Universal Robots PolyScope program: shot_03_120.urp

Program shot_03_120 (installation=default createdIn=5.11.11 lastSavedIn=5.11.11)
Robot Program (runOnlyOnce=true)
  Script file shot_03_120.script
    | def Program():
    |   CameraTcp = p[0.035, 0, 0.11, 1.2092, 1.2092, 1.2092]
    |   CameraWeight = 2
    |   CameraCog = [0.035, 0, 0.11]
    |   DefaultSpeed = 0.1
    |   DefaultZone = 0
    |   popup("Press 'Continue' to reset to Pose 0.", title="Ready?", blocking=True)
    |   set_tcp(CameraTcp)
    |   set_payload(CameraWeight, CameraCog)
    |   movej([2.8226, -1.6266, 1.8169, -1.6385, -1.6035, -2.1032], a=3.1416, v=0.3142, r=DefaultZone)
    |   popup("Press 'Continue' to go to Pose 1.", title="Pose 1", blocking=True)
    |   movel(p[0.49415, -0.01566, 0.29143, -1.3823, 1.14255, -0.9654], a=1, v=DefaultSpeed, r=DefaultZone)
    |   popup("Press 'Continue' to go to Pose 2.", title="Pose 2", blocking=True)
    |   movel(p[0.51704, -0.03671, 0.30239, -1.39572, 1.13007, -0.9443], a=1, v=DefaultSpeed, r=DefaultZone)
    |   popup("Press 'Continue' to go to Pose 3.", title="Pose 3", blocking=True)
    |   movel(p[0.5564, -0.0716, 0.32123, -1.41819, 1.10773, -0.90784], a=1, v=DefaultSpeed, r=DefaultZone)
    |   popup("Press 'Continue' to go to Pose 4.", title="Pose 4", blocking=True)
    |   movel(p[0.60924, -0.11494, 0.34645, -1.4463, 1.07643, -0.85942], a=1, v=DefaultSpeed, r=DefaultZone)
    |   popup("Press 'Continue' to go to Pose 5.", title="Pose 5", blocking=True)
    |   movel(p[0.6663, -0.15398, 0.37355, -1.47245, 1.04299, -0.8105], a=1, v=DefaultSpeed, r=DefaultZone)
    |   popup("Press 'Continue' to go to Pose 6.", title="Pose 6", blocking=True)
    |   movel(p[0.71252, -0.1708, 0.39523, -1.48621, 1.0213, -0.78118], a=1, v=DefaultSpeed, r=DefaultZone)
    |   popup("Press 'Continue' to go to Pose 7.", title="Pose 7", blocking=True)
    |   movel(p[0.73552, -0.15426, 0.40545, -1.47934, 1.02256, -0.78869], a=1, v=DefaultSpeed, r=DefaultZone)
    |   popup("Press 'Continue' to go to Pose 8.", title="Pose 8", blocking=True)
    |   movel(p[0.74329, -0.12347, 0.40637, -1.45997, 1.03461, -0.81638], a=1, v=DefaultSpeed, r=DefaultZone)
    |   popup("Press 'Continue' to go to Pose 9.", title="Pose 9", blocking=True)
    |   movel(p[0.74266, -0.0907, 0.40168, -1.43528, 1.04897, -0.85068], a=1, v=DefaultSpeed, r=DefaultZone)
    |   popup("Press 'Continue' to go to Pose 10.", title="Pose 10", blocking=True)
    |   movel(p[0.73762, -0.06054, 0.39451, -1.40991, 1.06259, -0.88473], a=1, v=DefaultSpeed, r=DefaultZone)
    |   popup("Press 'Continue' to go to Pose 11.", title="Pose 11", blocking=True)
    |   movel(p[0.73124, -0.0355, 0.38717, -1.38733, 1.07389, -0.91407], a=1, v=DefaultSpeed, r=DefaultZone)
    |   popup("Press 'Continue' to go to Pose 12.", title="Pose 12", blocking=True)
    |   movel(p[0.7254, -0.0165, 0.38095, -1.36942, 1.08234, -0.93672], a=1, v=DefaultSpeed, r=DefaultZone)
    |   popup("Press 'Continue' to go to Pose 13.", title="Pose 13", blocking=True)
    |   movel(p[0.721, -0.00356, 0.37646, -1.35683, 1.08797, -0.95229], a=1, v=DefaultSpeed, r=DefaultZone)
    |   popup("Press 'Continue' to go to Pose 14.", title="Pose 14", blocking=True)
    |   movel(p[0.71839, 0.00374, 0.37383, -1.34952, 1.09105, -0.96114], a=1, v=DefaultSpeed, r=DefaultZone)
    |   popup("Press 'Continue' to go to Pose 15.", title="Pose 15", blocking=True)
    |   movel(p[0.71755, 0.00603, 0.373, -1.34706, 1.09188, -0.96399], a=1, v=DefaultSpeed, r=DefaultZone)
    |   popup("Press 'Continue' to go to Pose 15.", title="Pose 15", blocking=True)
    | end
    | 
    | Program()
